FUNCTION_BLOCK DELETAR
  (* Standard: 61499-2 *)
  (* Version 03-07-12, GASR *)
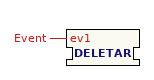
  EVENT_INPUT
    ev1;
  END_EVENT
END_FUNCTION_BLOCK
